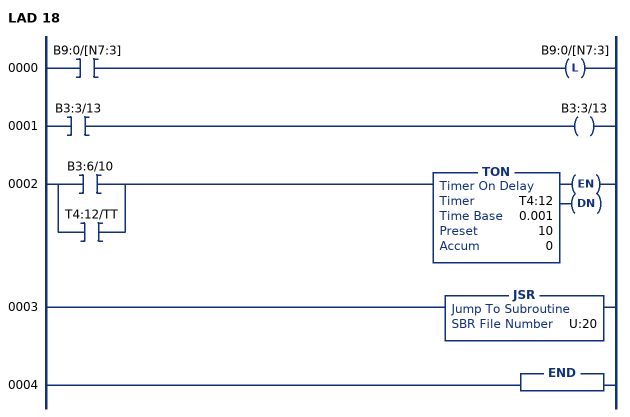
% Rung: 0 %
SOR XIC B9:0/[N7:3] OTL B9:0/[N7:3] EOR
% Rung: 1 %
SOR XIC B3:3/13 OTE B3:3/13 EOR
% Rung: 2 %
SOR BST XIC B3:6/10 NXB XIC T4:12/TT BND TON T4:12 0.001 10 0 EOR
% Rung: 3 %
SOR JSR U:20 EOR
% Rung: 4 %
SOR END EOR

LADDER 20
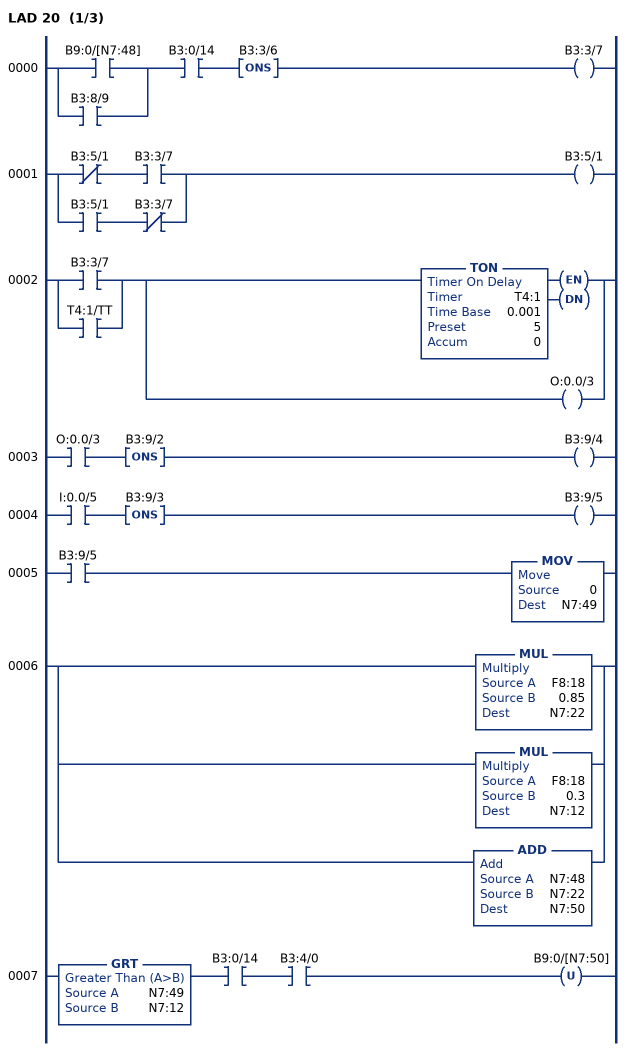
% Rung: 0 %
SOR BST XIC B9:0/[N7:48] NXB XIC B3:8/9 BND XIC B3:0/14 ONS B3:3/6 OTE B3:3/7 EOR
% Rung: 1 %
SOR BST XIO B3:5/1 XIC B3:3/7 NXB XIC B3:5/1 XIO B3:3/7 BND OTE B3:5/1 EOR
% Rung: 2 %
SOR BST XIC B3:3/7 NXB XIC T4:1/TT BND BST TON T4:1 0.001 5 0 NXB OTE O:0.0/3 BND EOR
% Rung: 3 %
SOR XIC O:0.0/3 ONS B3:9/2 OTE B3:9/4 EOR
% Rung: 4 %
SOR XIC I:0.0/5 ONS B3:9/3 OTE B3:9/5 EOR
% Rung: 5 %
SOR XIC B3:9/5 MOV 0 N7:49 EOR
% Rung: 6 %
SOR BST MUL F8:18 0.85 N7:22 NXB MUL F8:18 0.3 N7:12 NXB ADD N7:48 N7:22 N7:50 BND EOR
% Rung: 7 %
SOR GRT N7:49 N7:12 XIC B3:0/14 XIC B3:4/0 OTU B9:0/[N7:50] EOR

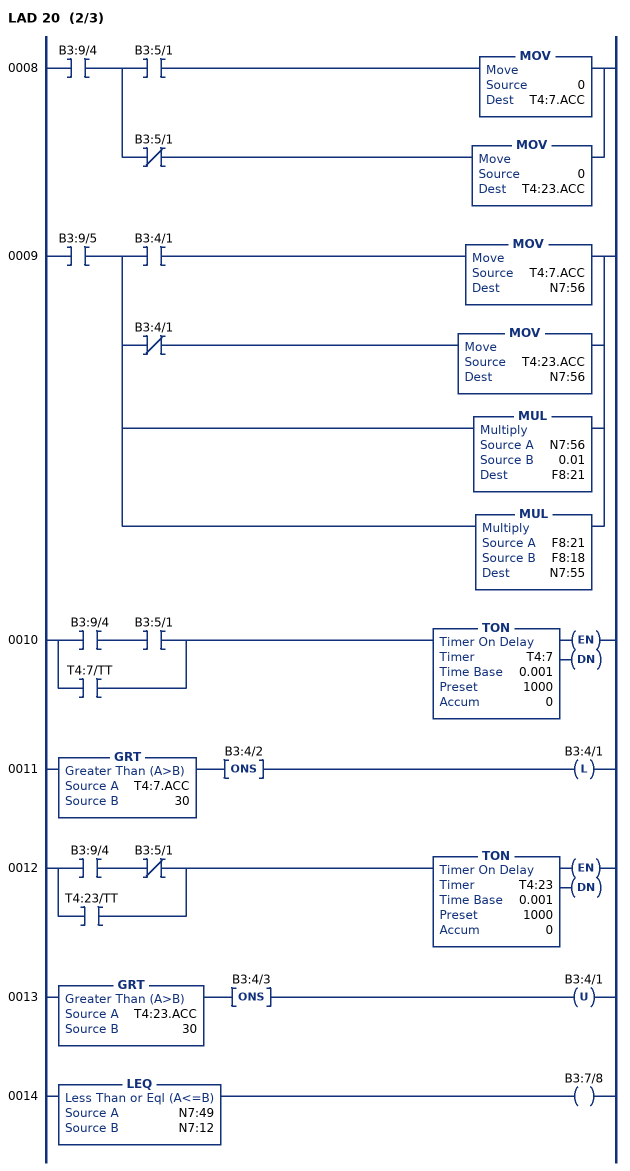
% Rung: 8 %
SOR XIC B3:9/4 BST XIC B3:5/1 MOV 0 T4:7.ACC NXB XIO B3:5/1 MOV 0 T4:23.ACC BND EOR
% Rung: 9 %
SOR XIC B3:9/5 BST XIC B3:4/1 MOV T4:7.ACC N7:56 NXB XIO B3:4/1 MOV T4:23.ACC N7:56 NXB MUL N7:56 0.01 F8:21 NXB MUL F8:21 F8:18 N7:55 BND EOR
% Rung: 10 %
SOR BST XIC B3:9/4 XIC B3:5/1 NXB XIC T4:7/TT BND TON T4:7 0.001 1000 0 EOR
% Rung: 11 %
SOR GRT T4:7.ACC 30 ONS B3:4/2 OTL B3:4/1 EOR
% Rung: 12 %
SOR BST XIC B3:9/4 XIO B3:5/1 NXB XIC T4:23/TT BND TON T4:23 0.001 1000 0 EOR
% Rung: 13 %
SOR GRT T4:23.ACC 30 ONS B3:4/3 OTU B3:4/1 EOR
% Rung: 14 %
SOR LEQ N7:49 N7:12 OTE B3:7/8 EOR

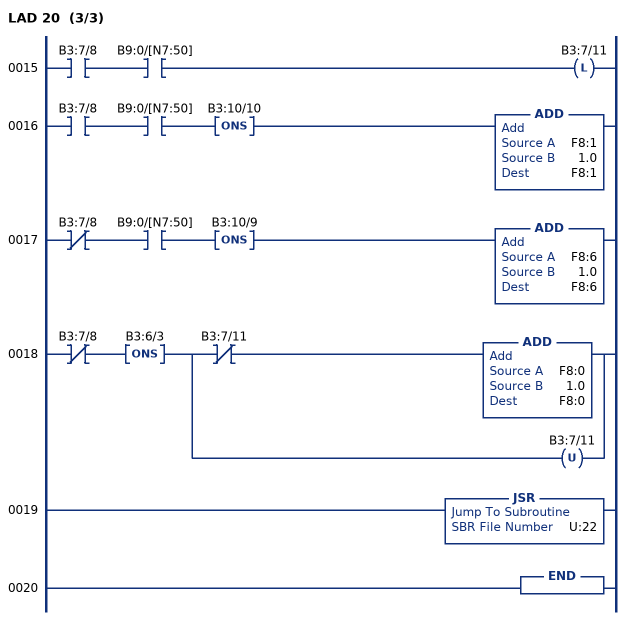
% Rung: 15 %
SOR XIC B3:7/8 XIC B9:0/[N7:50] OTL B3:7/11 EOR
% Rung: 16 %
SOR XIC B3:7/8 XIC B9:0/[N7:50] ONS B3:10/10 ADD F8:1 1.0 F8:1 EOR
% Rung: 17 %
SOR XIO B3:7/8 XIC B9:0/[N7:50] ONS B3:10/9 ADD F8:6 1.0 F8:6 EOR
% Rung: 18 %
SOR XIO B3:7/8 ONS B3:6/3 BST XIO B3:7/11 ADD F8:0 1.0 F8:0 NXB OTU B3:7/11 BND EOR
% Rung: 19 %
SOR JSR U:22 EOR
% Rung: 20 %
SOR END EOR

LADDER 22
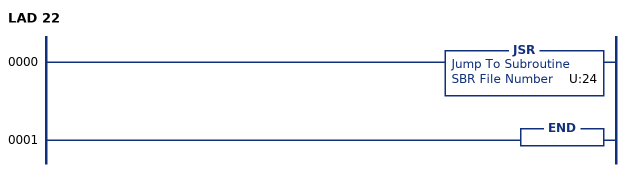
% Rung: 0 %
SOR JSR U:24 EOR
% Rung: 1 %
SOR END EOR

LADDER 24
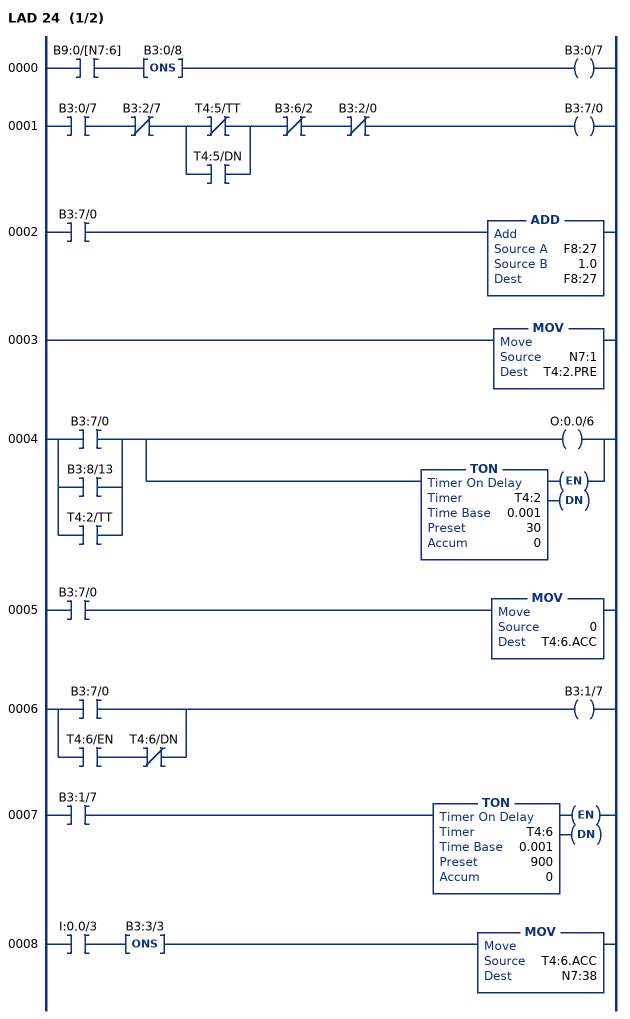
% Rung: 0 %
SOR XIC B9:0/[N7:6] ONS B3:0/8 OTE B3:0/7 EOR
% Rung: 1 %
SOR XIC B3:0/7 XIO B3:2/7 BST XIO T4:5/TT NXB XIC T4:5/DN BND XIO B3:6/2 XIO B3:2/0 OTE B3:7/0 EOR
% Rung: 2 %
SOR XIC B3:7/0 ADD F8:27 1.0 F8:27 EOR
% Rung: 3 %
SOR MOV N7:1 T4:2.PRE EOR
% Rung: 4 %
SOR BST XIC B3:7/0 NXB XIC B3:8/13 NXB XIC T4:2/TT BND BST OTE O:0.0/6 NXB TON T4:2 0.001 30 0 BND EOR
% Rung: 5 %
SOR XIC B3:7/0 MOV 0 T4:6.ACC EOR
% Rung: 6 %
SOR BST XIC B3:7/0 NXB XIC T4:6/EN XIO T4:6/DN BND OTE B3:1/7 EOR
% Rung: 7 %
SOR XIC B3:1/7 TON T4:6 0.001 900 0 EOR
% Rung: 8 %
SOR XIC I:0.0/3 ONS B3:3/3 MOV T4:6.ACC N7:38 EOR

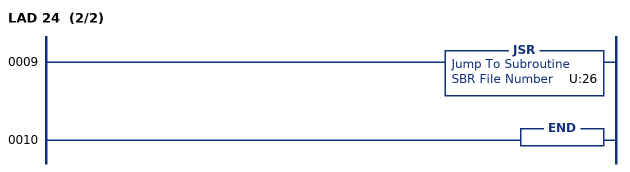
% Rung: 9 %
SOR JSR U:26 EOR
% Rung: 10 %
SOR END EOR

LADDER 26
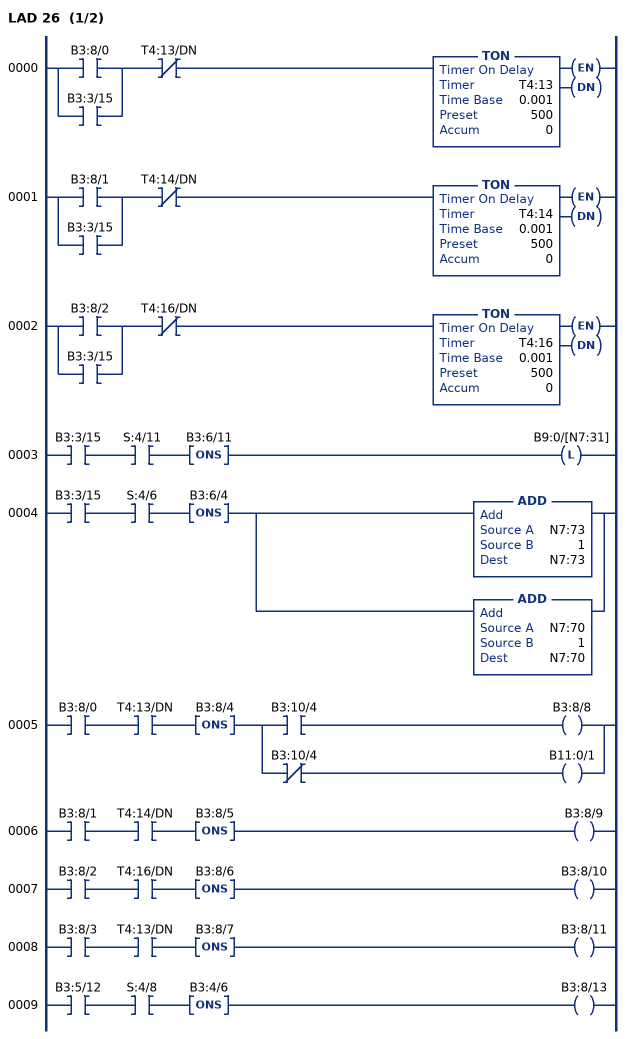
% Rung: 0 %
SOR BST XIC B3:8/0 NXB XIC B3:3/15 BND XIO T4:13/DN TON T4:13 0.001 500 0 EOR
% Rung: 1 %
SOR BST XIC B3:8/1 NXB XIC B3:3/15 BND XIO T4:14/DN TON T4:14 0.001 500 0 EOR
% Rung: 2 %
SOR BST XIC B3:8/2 NXB XIC B3:3/15 BND XIO T4:16/DN TON T4:16 0.001 500 0 EOR
% Rung: 3 %
SOR XIC B3:3/15 XIC S:4/11 ONS B3:6/11 OTL B9:0/[N7:31] EOR
% Rung: 4 %
SOR XIC B3:3/15 XIC S:4/6 ONS B3:6/4 BST ADD N7:73 1 N7:73 NXB ADD N7:70 1 N7:70 BND EOR
% Rung: 5 %
SOR XIC B3:8/0 XIC T4:13/DN ONS B3:8/4 BST XIC B3:10/4 OTE B3:8/8 NXB XIO B3:10/4 OTE B11:0/1 BND EOR
% Rung: 6 %
SOR XIC B3:8/1 XIC T4:14/DN ONS B3:8/5 OTE B3:8/9 EOR
% Rung: 7 %
SOR XIC B3:8/2 XIC T4:16/DN ONS B3:8/6 OTE B3:8/10 EOR
% Rung: 8 %
SOR XIC B3:8/3 XIC T4:13/DN ONS B3:8/7 OTE B3:8/11 EOR
% Rung: 9 %
SOR XIC B3:5/12 XIC S:4/8 ONS B3:4/6 OTE B3:8/13 EOR

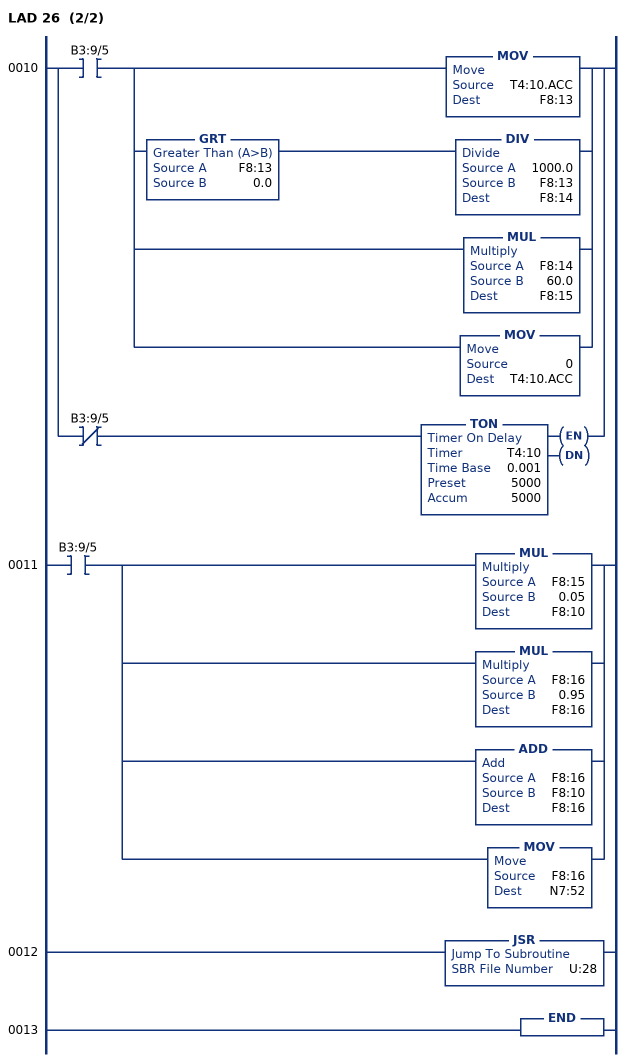
% Rung: 10 %
SOR BST XIC B3:9/5 BST MOV T4:10.ACC F8:13 NXB GRT F8:13 0.0 DIV 1000.0 F8:13 F8:14 NXB MUL F8:14 60.0 F8:15 NXB MOV 0 T4:10.ACC BND NXB XIO B3:9/5 TON T4:10 0.001 5000 5000 BND EOR
% Rung: 11 %
SOR XIC B3:9/5 BST MUL F8:15 0.05 F8:10 NXB MUL F8:16 0.95 F8:16 NXB ADD F8:16 F8:10 F8:16 NXB MOV F8:16 N7:52 BND EOR
% Rung: 12 %
SOR JSR U:28 EOR
% Rung: 13 %
SOR END EOR

LADDER 28
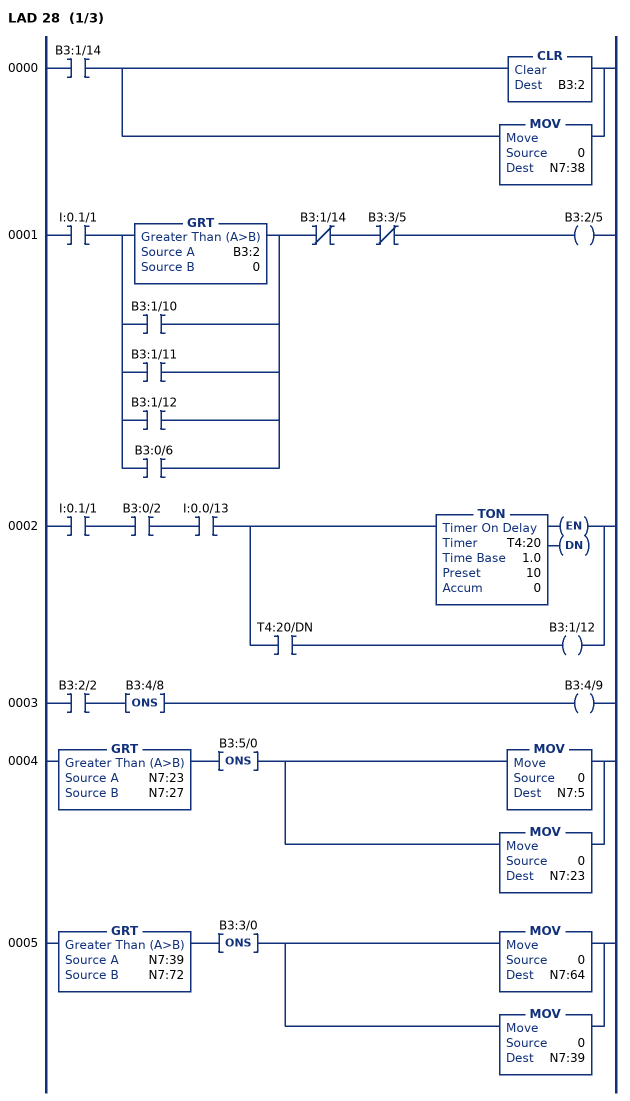
% Rung: 0 %
SOR XIC B3:1/14 BST CLR B3:2 NXB MOV 0 N7:38 BND EOR
% Rung: 1 %
SOR XIC I:0.1/1 BST GRT B3:2 0 NXB XIC B3:1/10 NXB XIC B3:1/11 NXB XIC B3:1/12 NXB XIC B3:0/6 BND XIO B3:1/14 XIO B3:3/5 OTE B3:2/5 EOR
% Rung: 2 %
SOR XIC I:0.1/1 XIC B3:0/2 XIC I:0.0/13 BST TON T4:20 1.0 10 0 NXB XIC T4:20/DN OTE B3:1/12 BND EOR
% Rung: 3 %
SOR XIC B3:2/2 ONS B3:4/8 OTE B3:4/9 EOR
% Rung: 4 %
SOR GRT N7:23 N7:27 ONS B3:5/0 BST MOV 0 N7:5 NXB MOV 0 N7:23 BND EOR
% Rung: 5 %
SOR GRT N7:39 N7:72 ONS B3:3/0 BST MOV 0 N7:64 NXB MOV 0 N7:39 BND EOR

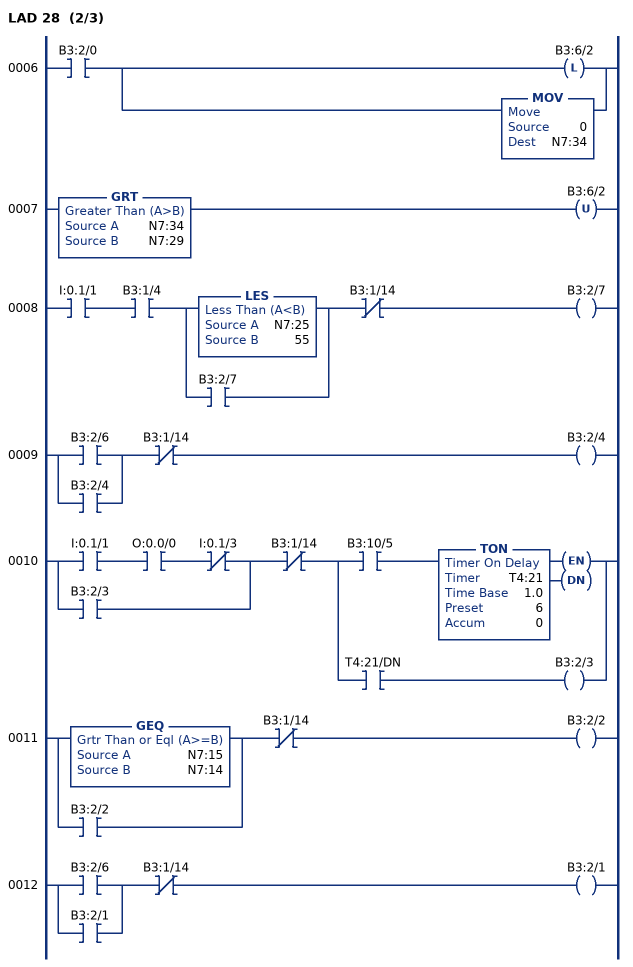
% Rung: 6 %
SOR XIC B3:2/0 BST OTL B3:6/2 NXB MOV 0 N7:34 BND EOR
% Rung: 7 %
SOR GRT N7:34 N7:29 OTU B3:6/2 EOR
% Rung: 8 %
SOR XIC I:0.1/1 XIC B3:1/4 BST LES N7:25 55 NXB XIC B3:2/7 BND XIO B3:1/14 OTE B3:2/7 EOR
% Rung: 9 %
SOR BST XIC B3:2/6 NXB XIC B3:2/4 BND XIO B3:1/14 OTE B3:2/4 EOR
% Rung: 10 %
SOR BST XIC I:0.1/1 XIC O:0.0/0 XIO I:0.1/3 NXB XIC B3:2/3 BND XIO B3:1/14 BST XIC B3:10/5 TON T4:21 1.0 6 0 NXB XIC T4:21/DN OTE B3:2/3 BND EOR
% Rung: 11 %
SOR BST GEQ N7:15 N7:14 NXB XIC B3:2/2 BND XIO B3:1/14 OTE B3:2/2 EOR
% Rung: 12 %
SOR BST XIC B3:2/6 NXB XIC B3:2/1 BND XIO B3:1/14 OTE B3:2/1 EOR

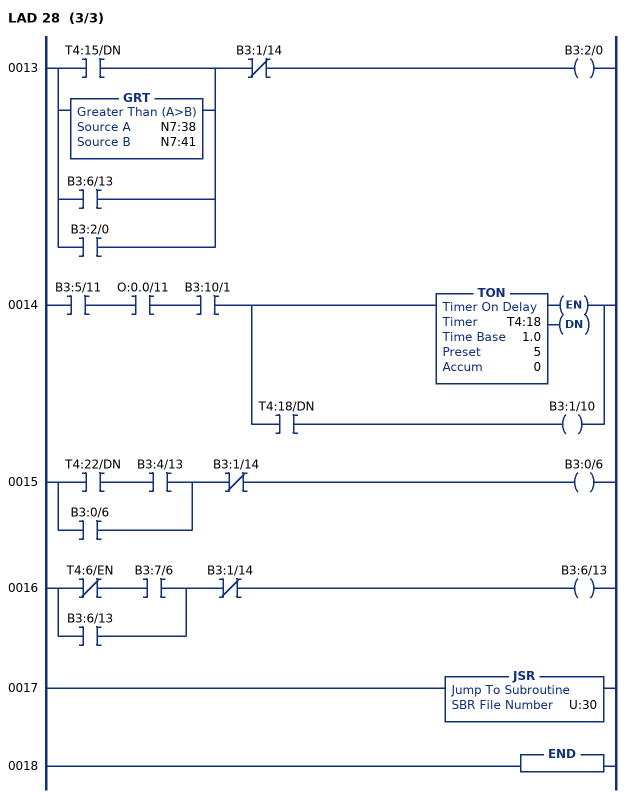
% Rung: 13 %
SOR BST XIC T4:15/DN NXB GRT N7:38 N7:41 NXB XIC B3:6/13 NXB XIC B3:2/0 BND XIO B3:1/14 OTE B3:2/0 EOR
% Rung: 14 %
SOR XIC B3:5/11 XIC O:0.0/11 XIC B3:10/1 BST TON T4:18 1.0 5 0 NXB XIC T4:18/DN OTE B3:1/10 BND EOR
% Rung: 15 %
SOR BST XIC T4:22/DN XIC B3:4/13 NXB XIC B3:0/6 BND XIO B3:1/14 OTE B3:0/6 EOR
% Rung: 16 %
SOR BST XIO T4:6/EN XIC B3:7/6 NXB XIC B3:6/13 BND XIO B3:1/14 OTE B3:6/13 EOR
% Rung: 17 %
SOR JSR U:30 EOR
% Rung: 18 %
SOR END EOR

LADDER 30
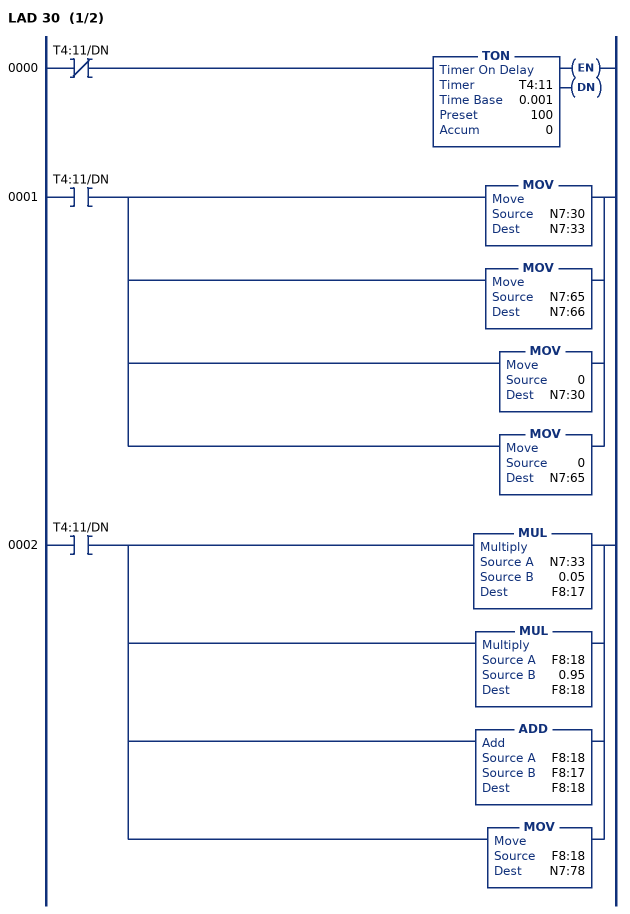
% Rung: 0 %
SOR XIO T4:11/DN TON T4:11 0.001 100 0 EOR
% Rung: 1 %
SOR XIC T4:11/DN BST MOV N7:30 N7:33 NXB MOV N7:65 N7:66 NXB MOV 0 N7:30 NXB MOV 0 N7:65 BND EOR
% Rung: 2 %
SOR XIC T4:11/DN BST MUL N7:33 0.05 F8:17 NXB MUL F8:18 0.95 F8:18 NXB ADD F8:18 F8:17 F8:18 NXB MOV F8:18 N7:78 BND EOR

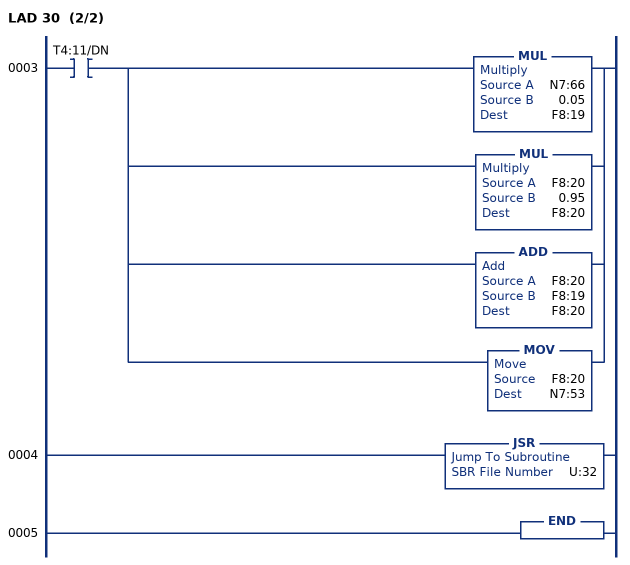
% Rung: 3 %
SOR XIC T4:11/DN BST MUL N7:66 0.05 F8:19 NXB MUL F8:20 0.95 F8:20 NXB ADD F8:20 F8:19 F8:20 NXB MOV F8:20 N7:53 BND EOR
% Rung: 4 %
SOR JSR U:32 EOR
% Rung: 5 %
SOR END EOR

LADDER 32
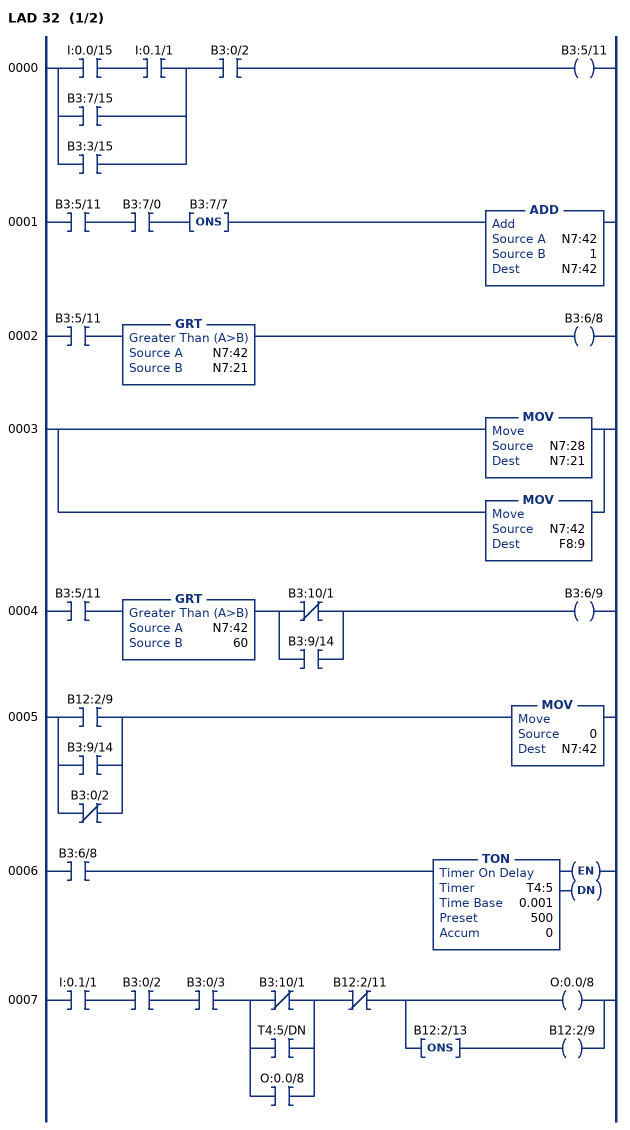
% Rung: 0 %
SOR BST XIC I:0.0/15 XIC I:0.1/1 NXB XIC B3:7/15 NXB XIC B3:3/15 BND XIC B3:0/2 OTE B3:5/11 EOR
% Rung: 1 %
SOR XIC B3:5/11 XIC B3:7/0 ONS B3:7/7 ADD N7:42 1 N7:42 EOR
% Rung: 2 %
SOR XIC B3:5/11 GRT N7:42 N7:21 OTE B3:6/8 EOR
% Rung: 3 %
SOR BST MOV N7:28 N7:21 NXB MOV N7:42 F8:9 BND EOR
% Rung: 4 %
SOR XIC B3:5/11 GRT N7:42 60 BST XIO B3:10/1 NXB XIC B3:9/14 BND OTE B3:6/9 EOR
% Rung: 5 %
SOR BST XIC B12:2/9 NXB XIC B3:9/14 NXB XIO B3:0/2 BND MOV 0 N7:42 EOR
% Rung: 6 %
SOR XIC B3:6/8 TON T4:5 0.001 500 0 EOR
% Rung: 7 %
SOR XIC I:0.1/1 XIC B3:0/2 XIC B3:0/3 BST XIO B3:10/1 NXB XIC T4:5/DN NXB XIC O:0.0/8 BND XIO B12:2/11 BST OTE O:0.0/8 NXB ONS B12:2/13 OTE B12:2/9 BND EOR

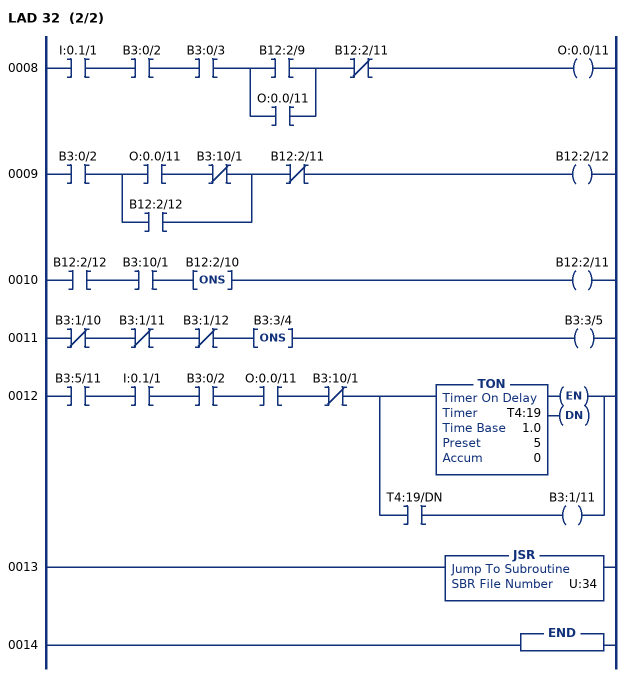
% Rung: 8 %
SOR XIC I:0.1/1 XIC B3:0/2 XIC B3:0/3 BST XIC B12:2/9 NXB XIC O:0.0/11 BND XIO B12:2/11 OTE O:0.0/11 EOR
% Rung: 9 %
SOR XIC B3:0/2 BST XIC O:0.0/11 XIO B3:10/1 NXB XIC B12:2/12 BND XIO B12:2/11 OTE B12:2/12 EOR
% Rung: 10 %
SOR XIC B12:2/12 XIC B3:10/1 ONS B12:2/10 OTE B12:2/11 EOR
% Rung: 11 %
SOR XIO B3:1/10 XIO B3:1/11 XIO B3:1/12 ONS B3:3/4 OTE B3:3/5 EOR
% Rung: 12 %
SOR XIC B3:5/11 XIC I:0.1/1 XIC B3:0/2 XIC O:0.0/11 XIO B3:10/1 BST TON T4:19 1.0 5 0 NXB XIC T4:19/DN OTE B3:1/11 BND EOR
% Rung: 13 %
SOR JSR U:34 EOR
% Rung: 14 %
SOR END EOR

LADDER 34
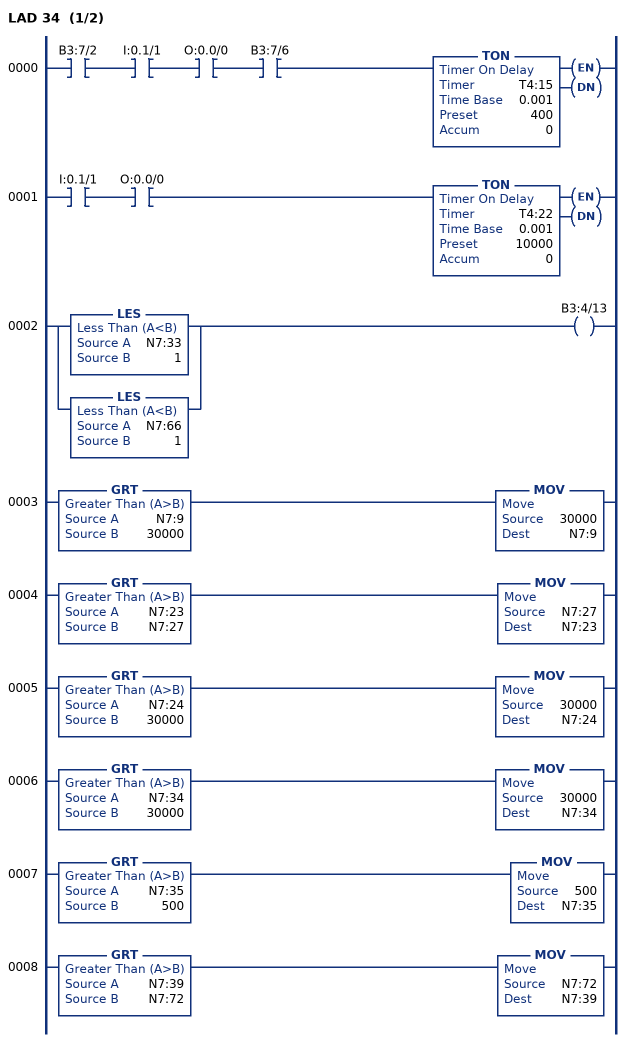
% Rung: 0 %
SOR XIC B3:7/2 XIC I:0.1/1 XIC O:0.0/0 XIC B3:7/6 TON T4:15 0.001 400 0 EOR
% Rung: 1 %
SOR XIC I:0.1/1 XIC O:0.0/0 TON T4:22 0.001 10000 0 EOR
% Rung: 2 %
SOR BST LES N7:33 1 NXB LES N7:66 1 BND OTE B3:4/13 EOR
% Rung: 3 %
SOR GRT N7:9 30000 MOV 30000 N7:9 EOR
% Rung: 4 %
SOR GRT N7:23 N7:27 MOV N7:27 N7:23 EOR
% Rung: 5 %
SOR GRT N7:24 30000 MOV 30000 N7:24 EOR
% Rung: 6 %
SOR GRT N7:34 30000 MOV 30000 N7:34 EOR
% Rung: 7 %
SOR GRT N7:35 500 MOV 500 N7:35 EOR
% Rung: 8 %
SOR GRT N7:39 N7:72 MOV N7:72 N7:39 EOR

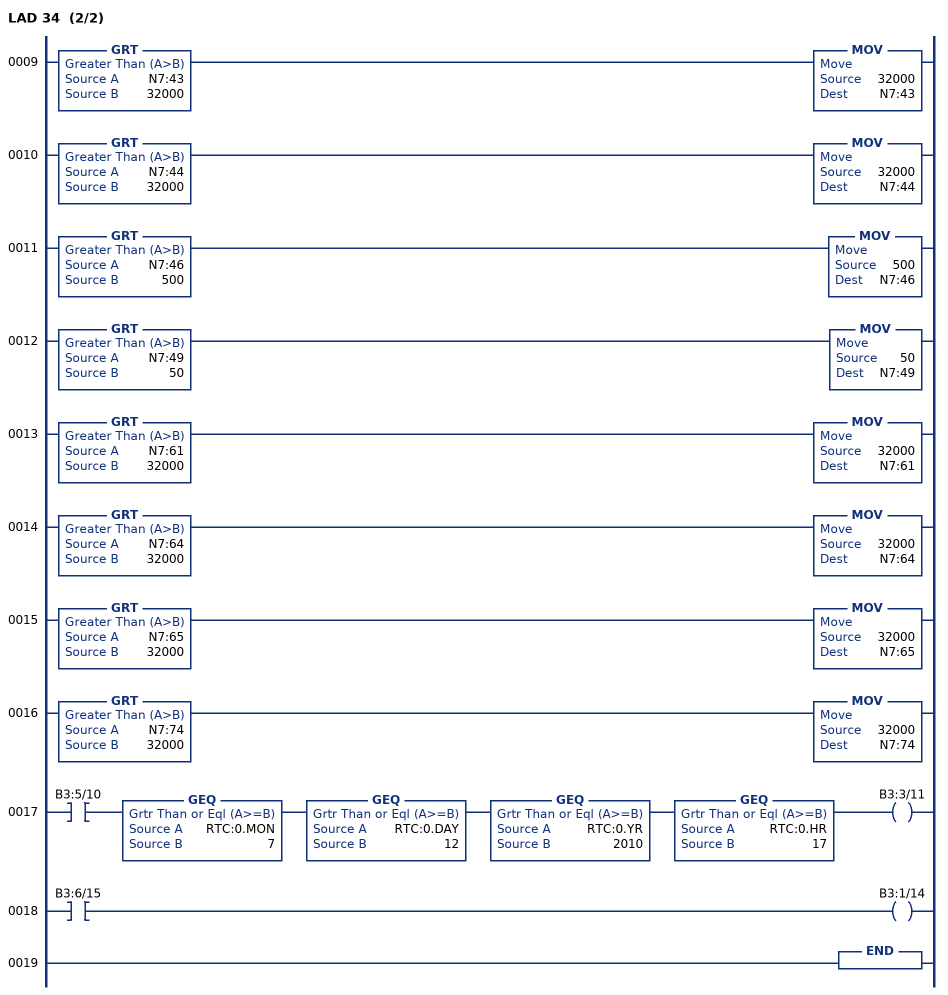
% Rung: 9 %
SOR GRT N7:43 32000 MOV 32000 N7:43 EOR
% Rung: 10 %
SOR GRT N7:44 32000 MOV 32000 N7:44 EOR
% Rung: 11 %
SOR GRT N7:46 500 MOV 500 N7:46 EOR
% Rung: 12 %
SOR GRT N7:49 50 MOV 50 N7:49 EOR
% Rung: 13 %
SOR GRT N7:61 32000 MOV 32000 N7:61 EOR
% Rung: 14 %
SOR GRT N7:64 32000 MOV 32000 N7:64 EOR
% Rung: 15 %
SOR GRT N7:65 32000 MOV 32000 N7:65 EOR
% Rung: 16 %
SOR GRT N7:74 32000 MOV 32000 N7:74 EOR
% Rung: 17 %
SOR XIC B3:5/10 GEQ RTC:0.MON 7 GEQ RTC:0.DAY 12 GEQ RTC:0.YR 2010 GEQ RTC:0.HR 17 OTE B3:3/11 EOR
% Rung: 18 %
SOR XIC B3:6/15 OTE B3:1/14 EOR
% Rung: 19 %
SOR END EOR

DATA TABLE (non-zero values as saved)
DATA B3
% B3:0 % 0X4014 0X0100 0X0000 0X4014 0X2C01 0X6AA8 0X4049 0X8026 0X0000 0X0000
% B3:10 % 0X0078 0X000E 0X0000 0X0400 0X0000 0X0000 0X0000 0X0000 0X0000 0X0000
DATA T4
% .PRE .ACC %
% T4:0 % 9 0
% T4:1 % 5 0
% T4:2 % 30 0
% T4:3 % 1000 0
% T4:4 % 50 0
% T4:5 % 500 0
% T4:6 % 900 0
% T4:7 % 1000 0
% T4:8 % 1000 0
% T4:9 % 16 0
% T4:10 % 5000 5000
% T4:11 % 100 0
% T4:12 % 10 0
% T4:13 % 500 0
% T4:14 % 500 0
% T4:15 % 400 0
% T4:16 % 500 0
% T4:17 % 1000 0
% T4:18 % 5 0
% T4:19 % 5 0
% T4:20 % 10 0
% T4:21 % 6 0
% T4:22 % 10000 0
% T4:23 % 1000 0
% T4:24 % 1000 0
% T4:25 % 250 250
DATA C5
% .PRE .ACC %
% C5:2 % 20 -16929
% C5:3 % 32000 0
% C5:4 % 32000 0
% C5:6 % 0 1513
% C5:7 % 0 1467
% C5:8 % 10000 47
% C5:9 % 1800 0
DATA R6
% .LEN .POS %
% R6:0 % 1200 0
% R6:1 % 600 0
% R6:2 % 1200 0
% R6:3 % 25 24
% R6:4 % 300 0
% R6:5 % 5 4
% R6:6 % 1000 0
% R6:7 % 300 0
% R6:8 % 600 0
DATA N7
% N7:0 % 748 30 5 811 1 0 1071 90 85 0
% N7:10 % 8 7 0 0 1500 0 30 579 45 15
% N7:20 % 0 4310 0 0 0 2 -398 33 4310 650
% N7:30 % 0 549 549 0 651 0 30 13 0 0
% N7:40 % 1155 300 0 32000 32000 0 500 748 846 50
% N7:50 % 846 64 90 0 26 27 66 0 1001 0
% N7:60 % 1 32000 154 15 32000 0 0 0 0 0
% N7:70 % 0 0 15 0 32000 0 126 0 0 0
% N7:80 % 0 0 0 501 0 0 0 0 0 0
DATA F8
% F8:0 % 1.677722e+07 1.677722e+07 6627153 1.677722e+07 3451002
% F8:5 % 1.677722e+07 1.677722e+07 1.677722e+07 1.677722e+07 0
% F8:10 % 0.6 0.093 25 5000 0.2
% F8:15 % 12 89.70184 0 0 0
% F8:20 % 0 0.66 0.64 0 0
% F8:25 % 1.487718e+07 1.677722e+07 1.677722e+07 0 0
DATA B9
% B9:70 % 0X0000 0X0000 0X0000 0X0000 0X0000 0X001F 0X0000 0XE010 0XFFBF 0XFFFF
% B9:80 % 0XFFFF 0XFFFF 0XFFFF 0XFFFF 0XFFFF 0XFEFF 0XFFFB 0XBFFF 0XFFFF 0XBFFF
% B9:90 % 0XFFFF 0XFFFF 0XFFFF 0XFFEB 0X73FF 0XFFDF 0XFFFF 0XFDFF 0X7FBF 0X7F7F
% B9:100 % 0XFFFB 0X77F7 0XBF7F 0XFB7F 0XF7F9 0XBDFF 0XFF96 0XDF67 0XEFFF 0XFFFE
% B9:110 % 0XFDDF 0XEFFF 0XBBFF 0XF7FD 0X7EFF 0XB357 0XFFBD 0XFBBC 0XD79F 0XFFFD
% B9:120 % 0X35DE 0XE7DE 0XF3EB 0X73F3 0XFE77 0XFEC7 0XF6FF 0X3DFE 0X8DB7 0X7DBB
% B9:130 % 0XFF9F 0XED7F 0XBD5E 0XEFAE 0XBB85 0X4DE7 0XFBF3 0XAE57 0X9CBC 0XF7F8
% B9:140 % 0X9567 0XE922 0XCCF9 0XE47F 0XF81D 0XCF4B 0XD693 0X3EAB 0X6957 0XB93F
% B9:150 % 0XFEBF 0XE2DA 0X2D5E 0XC2A8 0XD274 0XEE7F 0X7FEF 0X4378 0X5711 0XBE3F
% B9:160 % 0XFD36 0XE0F7 0XDD86 0X8A6C 0XF33C 0XBBFF 0X27EC 0X4C5F 0X2C8C 0XB290
% B9:170 % 0XC16C 0XE29B 0XA45B 0X6E4C 0X226D 0XF4DC 0XB264 0X8A40 0XBE56 0X4F7E
% B9:180 % 0XFCE7 0X5BD1 0X87DB 0X0065 0XB795 0XD426 0XCF52 0X1CCC 0X36F6 0X2442
% B9:190 % 0XE39B 0X413B 0X50B8 0X49CE 0X5510 0X2C0A 0X38C3 0X5206 0X7C82 0X4CE2
% B9:200 % 0X6885 0X8324 0X9421 0XAFD0 0X9AE1 0X050F 0X5008 0XBAA0 0X128F 0X1480
% B9:210 % 0X4941 0X982F 0X2EC1 0X508F 0X4418 0X2D10 0XADA0 0X0126 0X1DA0 0X1BFA
% B9:220 % 0X4194 0X10EA 0X2E02 0X9220 0X5251 0X3085 0X2600 0X38E2 0X8002 0X0224
% B9:230 % 0X4385 0X80A4 0X085D 0X0005 0XA411 0X00B4 0XA114 0X1049 0X4B00 0X6042
% B9:240 % 0X0845 0X10A6 0X0223 0X0048 0X3242 0X8016 0X0041 0X0942 0X5102 0X0341
% B9:250 % 0X22D0 0X0140 0X0800 0X5810 0X0400 0X815C
DATA B11
% B11:80 % 0X0000 0X0000 0X0000 0X0428 0X0010 0X0000 0X0000 0X0020 0X0400 0X4040
% B11:90 % 0X0001 0X0010 0X0002 0X0850 0X0000 0X0004 0X0500 0X0400 0X4000 0X2000
% B11:100 % 0X0000 0X0000 0X0000 0X0200 0X0000 0X4000 0X0204 0X0400 0X9000 0X8000
% B11:110 % 0X8040 0X0101 0X0000 0X1000 0X5108 0X3040 0X0101 0X0000 0X0000 0X0060
% B11:120 % 0X0820 0X0000 0X0040 0X0200 0X0841 0X0000 0X0000 0X0001 0X0100 0X0000
% B11:130 % 0X0202 0X4004 0X0000 0X0001 0X0000 0X0000 0X0000 0X0000 0X0201 0X0400
% B11:140 % 0X0004 0X8082 0X0000 0X0200 0XC000 0X0000 0X0048 0X0000 0X0600 0X0000
% B11:150 % 0X4100 0X8000 0X0000 0X0000 0X1000 0X0000 0X0800 0X0020 0X0000 0X0012
% B11:160 % 0X0080 0X0000 0X0000 0X0100 0X0100 0X0000 0X0400 0X0014 0X0000 0X0002
% B11:170 % 0X0000 0X0000 0X0000 0X0080 0X04A8 0X0000 0X0000 0X0000 0X0008 0X0000
% B11:180 % 0X0000 0X0000 0X0000 0X1080 0X0000 0X0000 0X0000 0X0020 0X0000 0X0000
% B11:190 % 0X8100 0X0000 0X0080 0X0000 0X0040 0X0001 0X0001 0X0040 0X0000 0X0000
% B11:200 % 0X0000 0X0000 0X0000 0X0000 0X0000 0X0000 0X0400 0X0000 0X0000 0X0400
% B11:210 % 0X0000 0X0000 0X0000 0X0000 0X0400 0X0000 0X2000 0X0000 0X0000 0X0000
% B11:220 % 0X0000 0X0011 0X4020 0X0020 0X0010 0X0000 0X0000 0X0000 0X0000 0X0200
% B11:230 % 0X0001 0X0000 0X0400 0X0000 0X0060 0X0000 0X0402 0X0000 0X8000 0X0400
% B11:240 % 0X0100 0X0000 0X0000 0X0000 0X0000 0X0000 0X0204 0X0800 0X0000 0X0000
% B11:250 % 0X2000 0X0000 0X0000 0X0000 0X0000 0X0000
DATA B12
% B12:0 % 0X0008 0X000C 0X0100
DATA B14
% B14:0 % 0X2000 0X0000 0X0400 0X0080 0X0000 0X0000 0X1000 0X0000 0X0000 0X0200
% B14:10 % 0X0800 0X0200 0X0000 0X0000 0X0000 0X0000 0X0008 0X1000 0X0080 0X0000
% B14:20 % 0X0000 0X0000 0X0202 0X0400 0X0040 0X0000 0X0000 0X0002 0X0000 0X0000
% B14:30 % 0X0001 0X0100 0X0000 0X0000 0X8000 0X8002 0X0000 0X0080 0X0000 0X0000
% B14:40 % 0X1000 0X0000 0X0000 0X0000 0X2500 0X0000 0X0004 0X0000 0X0802 0X0040
% B14:50 % 0X0021 0X0000 0X0000 0X0000 0X0020 0X0100 0X0000 0X0000 0X0000 0X0000
% B14:60 % 0X0100 0X0000 0X0000 0X0000 0X0000 0X0400 0X0000 0X0000 0X0000 0X0400
% B14:70 % 0X0200 0X0800 0X0200 0X0000 0X0000 0X0000 0X0000 0X0000 0X0008 0X0000
% B14:80 % 0X0000 0XA001 0X0008 0X0000 0X0000 0X0000 0X0010 0X0000 0X8400 0X0000
% B14:90 % 0X2000 0X2000 0X2000 0X0000 0X0000 0X0000 0X0000 0X0000 0X0000 0X0000
% B14:100 % 0X0000 0X0100 0X0000 0X0000 0X0030 0X0000 0X0000 0X0000 0X0000 0X0000
% B14:110 % 0X0000 0X0000 0X0280 0X0000 0X0000 0X0000 0X0000 0X0000 0X0000 0X0000
% B14:120 % 0X0000 0X0000 0X0000 0X0000 0X2000 0X0000 0X0000 0X0200 0X0000 0X0000
% B14:130 % 0X0008 0X0820 0X0000 0X0000 0X0000 0X0000 0X0000 0X0000 0X0000 0X0000
% B14:140 % 0X0000 0X0000 0X0000 0X0000 0X0002 0X0000 0X0100 0X0004 0X0000 0X0000
% B14:150 % 0X000C 0X0000 0X0100 0X0000 0X4000 0X0000 0X0040 0X0000 0X0000 0X0000
% B14:160 % 0X0000 0X0000 0X0000 0X0000 0X0000 0X4000 0X0004 0X0000 0X0000 0X0008
% B14:170 % 0X0000 0X0000 0X0000 0X0000 0X0000 0X0000 0X0010 0X0000 0X0000 0X0000
% B14:180 % 0X0000 0X0020 0X0000 0X0000 0X0300 0X0000 0X0000 0X0000 0X0080 0X0000
% B14:190 % 0X0000 0X0000 0X2000 0X0002 0X0000 0X0000 0X0400 0X0000 0X0000 0X0000
% B14:200 % 0X0000 0X0000 0X0000 0X0010 0X0000 0X0480 0X0000 0X0000 0X0000 0X0000
% B14:210 % 0X0000 0X0000 0X0000 0X0000 0X4000 0X0000 0X0000 0X0000 0X0000 0X0000
% B14:220 % 0X0000 0X0000 0X0000 0X0000 0X0000 0X4000 0X0000 0X0000 0X0000 0X0000
% B14:230 % 0X0804 0X0000 0X0002 0X0040 0X0000 0X0000 0X0000 0X0000 0X0000 0X0000
% B14:240 % 0X0000 0X0020 0X0000 0X0180 0X0000 0X0000 0X0000 0X0002 0X0000 0X0000
% B14:250 % 0X0000 0X0000 0X0080 0X0082 0X0020 0X0000
DATA N16
% N16:0 % 126 6 68 65 0 0 361 0 0 0
% N16:10 % 4096 0 0 267
DATA N17
% N17:0 % 512 0 0 0 0 0 125 0 17171 384
% N17:10 % 315 365 123
DATA B18
% B18:0 % 0X0000 0X0000 0X0000 0X8004 0X0000 0X0000 0X0000 0X0000 0X0000 0X8000
% B18:10 % 0X0000 0X000E 0X8000 0X0400 0X0000 0X0001 0X0000 0X0000 0X0000 0X0000
% B18:20 % 0X0800 0X0000 0X0000 0X0000 0X0000 0X0000 0X0001 0X0100 0X0000 0X0000
% B18:30 % 0X0000 0X0000 0X0000 0X0000 0X0000 0X0000 0X0000 0X0010 0X0000 0X0000
% B18:40 % 0X0000 0X0000 0X0000 0X0000 0X0080 0X4000 0X0000 0X0000 0X0000 0X0002
% B18:50 % 0X0000 0X0000 0X0000 0X0001 0X0008 0X0000 0X0400 0X1100 0X0000 0X0000
% B18:60 % 0X0000 0X0000 0X0000 0X0000 0X0204 0X0000 0X0000 0X0000 0X0000 0X0480
% B18:70 % 0X0000 0X4000 0X0000 0X0000 0X0020 0X0010 0X0000 0X0000 0X0000 0X0000
% B18:80 % 0X0200 0X0000 0X0000 0X0000 0X0000 0X0000 0X0000 0X0000 0X0000 0X0000
% B18:90 % 0X0000 0X0000 0X0000 0X2000 0X0080 0X0000 0X0000 0X0000 0X0000 0X0000
% B18:110 % 0X0000 0X4000 0X0002 0X0000 0X0002 0X0000 0X0002 0X0080 0X0000 0X0000
% B18:120 % 0X0000 0X0000 0X0004 0X0000 0X0000 0X0000 0X0000 0X0000 0X0000 0X0000
% B18:130 % 0X0000 0X0000 0X0000 0X0000 0X0000 0X0000 0X0000 0X0000 0X2800 0X0000
% B18:140 % 0X0000 0X0000 0X0000 0X0000 0X0000 0X0000 0X2000 0X0000 0X0020 0X0000
% B18:150 % 0X0000 0X2000 0X0000 0X0000 0X0020 0X0400 0X0000 0X0100 0X0000 0X0000
% B18:160 % 0X0000 0X0000 0X0000 0X0000 0X0000 0X0000 0X0020 0X0000 0X0000 0X0000
% B18:170 % 0X0000 0X0000 0X2000 0X0100 0X0000 0X0000 0X0000 0XD880 0X0067 0X0000
DATA F19
% F19:0 % 0 0 0 0 764534
DATA T20
% .PRE .ACC %
% T20:0 % 5 0
% T20:2 % 1000 0
% T20:4 % 5000 5000
% T20:5 % 5 0
% T20:7 % 5 0
% T20:10 % 5 0
% T20:11 % 5 0
% T20:12 % 300 0
DATA R21
% .LEN .POS %
% R21:0 % 1300 0
% R21:1 % 1000 0
% R21:2 % 1300 0
% R21:3 % 1000 0
DATA N24
% N24:0 % 1 1 1 1 0 0 0 0 0 0
% N24:10 % 0 1 1 1 1 1 1 1 1 1
% N24:20 % 1 1 1 1 1 1 1 1 1 1
% N24:30 % 1 1 1 1 1 1 1 1 1 1
% N24:40 % 1 1 1 1 1 1 1 1 1 0
% N24:50 % 0 0 0 0 1 1 1 1 1 1
% N24:60 % 1 1 1 1 1 1 1 1 1 1
% N24:70 % 1 1 1 1 1 1 1 1 1 1
% N24:80 % 1 1 1 1 1 1 1 1 1 1
% N24:90 % 1 1 1 1 1 1 1 1 1 1
% N24:100 % 1 1 1 1 1 1 1 1 1 1
% N24:110 % 1 1 1 1 1 1 1 1 1 1
% N24:120 % 1 1 1 0 0 0 0 0
